% RSLogix 500 project ladder do controle da valvula em malha aberta para o teste de degrau.RSS, saved by version 7.00.00.19 %
PROJECT "UNTITLED"    % processor: MicroLogix 1200 %

PROGRAM FILES
  LAD 2   4 rungs

DATA FILES
  O0 OUTPUT  7 elements
  I1 INPUT  10 elements
  S2 STATUS  66 elements
  B3 BINARY  1 elements
  T4 TIMER  1 elements
  C5 COUNTER  1 elements
  R6 CONTROL  1 elements
  N7 INTEGER  1 elements
  F8 FLOAT  3 elements

LADDER 2
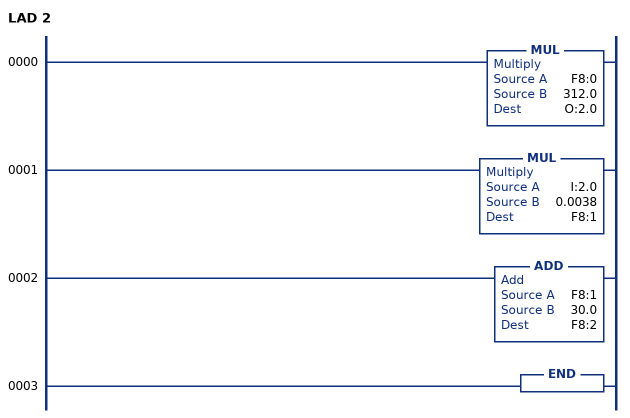
% Rung: 0 %
SOR MUL F8:0 312.0 O:2.0 EOR
% Rung: 1 %
SOR MUL I:2.0 0.0038 F8:1 EOR
% Rung: 2 %
SOR ADD F8:1 30.0 F8:2 EOR
% Rung: 3 %
SOR END EOR

DATA TABLE (non-zero values as saved)
DATA F8
% F8:0 % 50 2.3104 32.3104
